PROGRAM AutomationLibrary
VAR
	OrderHandling_Global: OrderHandling;
	mxErrorCodeOrder: INT;
	AGVControlSystem_GLobal: AGVControlSystem;
	RobotControlSystem_Global: RobotControlSystem;
	ABBGotoHome_TEST: ABBGotoHome;
	mxEnable: BOOL;
	BookingSystem_Global: BookingSystem;
	mxBookingDone: BOOL;
	mxBookingError: BOOL;
END_VAR

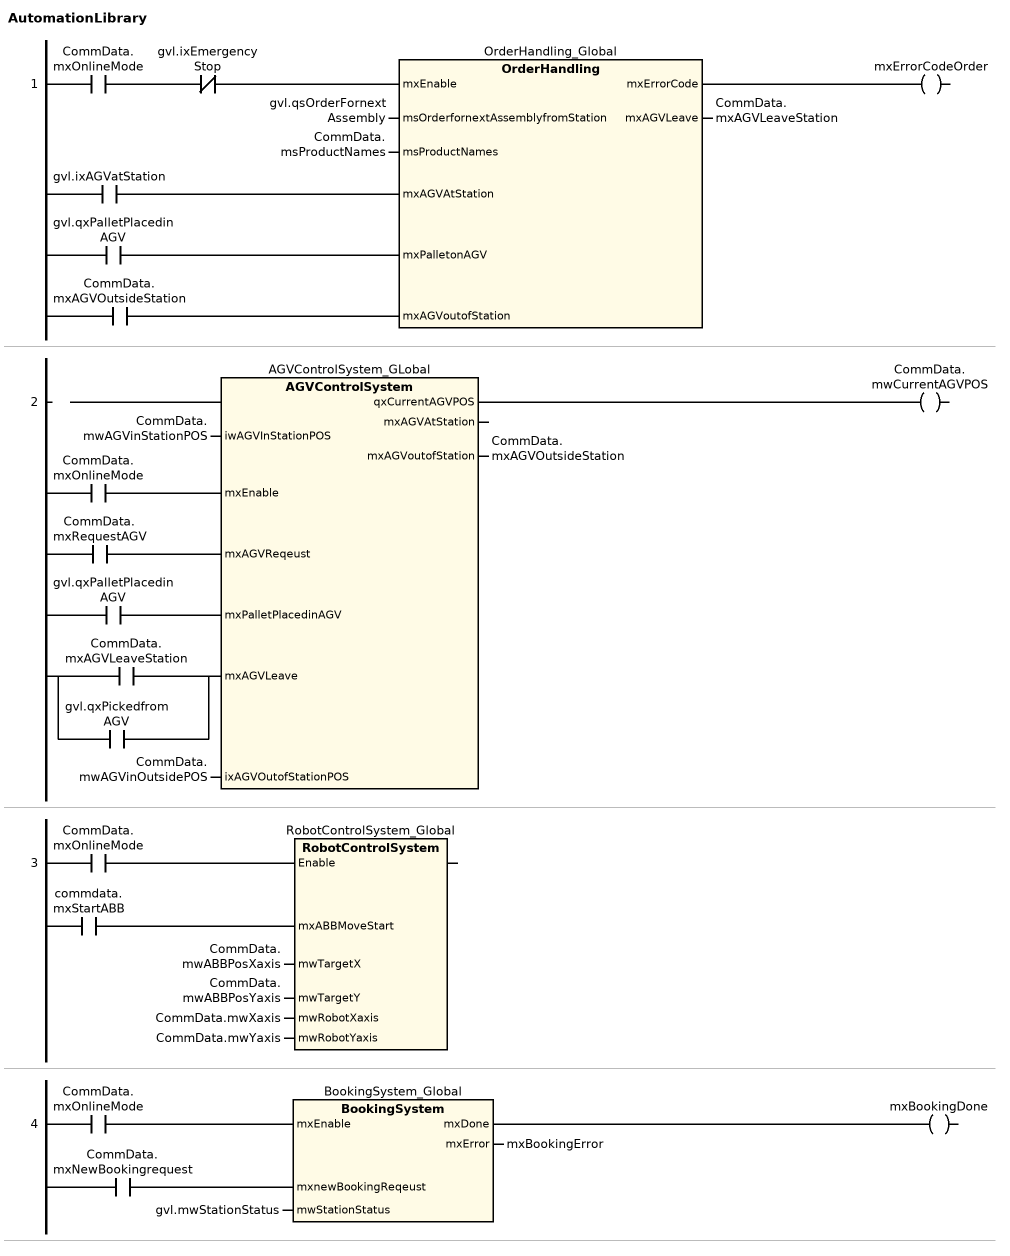
// NETWORK 1
OrderHandling_Global(
    mxEnable := CommData.mxOnlineMode AND NOT gvl.ixEmergencyStop,
    msOrderfornextAssemblyfromStation := gvl.qsOrderFornextAssembly,
    msProductNames := CommData.msProductNames,
    mxAGVAtStation := gvl.ixAGVatStation,
    mxPalletonAGV := gvl.qxPalletPlacedinAGV,
    mxAGVoutofStation := CommData.mxAGVOutsideStation,
    mxAGVLeave => CommData.mxAGVLeaveStation); // OrderHandling
mxErrorCodeOrder := OrderHandling_Global.mxErrorCode;

// NETWORK 2
AGVControlSystem_GLobal(
    iwAGVInStationPOS := CommData.mwAGVinStationPOS,
    mxEnable := CommData.mxOnlineMode,
    mxAGVReqeust := CommData.mxRequestAGV,
    mxPalletPlacedinAGV := gvl.qxPalletPlacedinAGV,
    mxAGVLeave := CommData.mxAGVLeaveStation OR gvl.qxPickedfromAGV,
    ixAGVOutofStationPOS := CommData.mwAGVinOutsidePOS,
    mxAGVoutofStation => CommData.mxAGVOutsideStation); // AGVControlSystem
CommData.mwCurrentAGVPOS := AGVControlSystem_GLobal.qxCurrentAGVPOS;

// NETWORK 3
RobotControlSystem_Global(
    Enable := CommData.mxOnlineMode,
    mxABBMoveStart := commdata.mxStartABB,
    mwTargetX := CommData.mwABBPosXaxis,
    mwTargetY := CommData.mwABBPosYaxis,
    mwRobotXaxis := CommData.mwXaxis,
    mwRobotYaxis := CommData.mwYaxis); // RobotControlSystem

// NETWORK 4
BookingSystem_Global(
    mxEnable := CommData.mxOnlineMode,
    mxnewBookingReqeust := CommData.mxNewBookingrequest,
    mwStationStatus := gvl.mwStationStatus,
    mxError => mxBookingError); // BookingSystem
mxBookingDone := BookingSystem_Global.mxDone;

END_PROGRAM

(* stored: Version 1.1.0.1, ProductVersion 3.1.4024.12
   POU AutomationLibrary: Id {77ab7955-b552-4839-b49a-3e1db13d0fe7}, SpecialFunc None *)
